{attribute 'qualified_only'}
VAR_GLOBAL PERSISTENT
	CantLiquidos:INT;
	CantPolvos:INT;
END_VAR

(* stored: Version 1.1.0.1, ProductVersion 3.1.4024.12
   GVL Configura: Id {c97b6783-d99e-4097-9a1f-edd73dc256cf} *)
